INTERFACE ITF_EM_Safety EXTENDS ITF_EM_Base

END_INTERFACE

(* stored: Version 1.1.0.1, ProductVersion 3.1.4024.10
   Itf ITF_EM_Safety: Id {13933a32-f04e-4a3e-b680-bdb10469a6c6} *)
